(* PLC project parallel.project, CODESYS CODESYS V3.5 SP17 Patch 3 *)
(* stored: creationDateTime 2022-06-05T18:18:27.6110924, modificationDateTime 2022-05-14T22:34:49.5278322 *)

PROGRAM flow_1

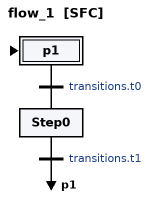
INITIAL_STEP p1:
END_STEP
TRANSITION FROM p1 TO Step0
  := transitions.t0;
END_TRANSITION
STEP Step0:
END_STEP
TRANSITION FROM Step0 TO p1
  := transitions.t1;
END_TRANSITION
END_PROGRAM

PROGRAM flow_2

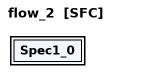
INITIAL_STEP Spec1_0:
END_STEP
END_PROGRAM

PROGRAM flow_3

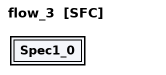
INITIAL_STEP Spec1_0:
END_STEP
END_PROGRAM

PROGRAM flow_4

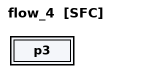
INITIAL_STEP p3:
END_STEP
END_PROGRAM

PROGRAM transitions

                  
                
END_PROGRAM

CONFIGURATION Application
  RESOURCE Application ON PLC
    VAR_GLOBAL  (* GVL *)
      t1 : BOOL;
      t3 : BOOL;
      t0 : BOOL;
      t2 : BOOL;
      t4 : BOOL;
    END_VAR
    TASK MainTask(INTERVAL := T#100ms, PRIORITY := 1);
    PROGRAM flow_1 WITH MainTask : flow_1;
    PROGRAM flow_2 WITH MainTask : flow_2;
    PROGRAM flow_3 WITH MainTask : flow_3;
    PROGRAM flow_4 WITH MainTask : flow_4;
  END_RESOURCE
END_CONFIGURATION
